Universal Robots PolyScope program: pick_place_robot_2.urp

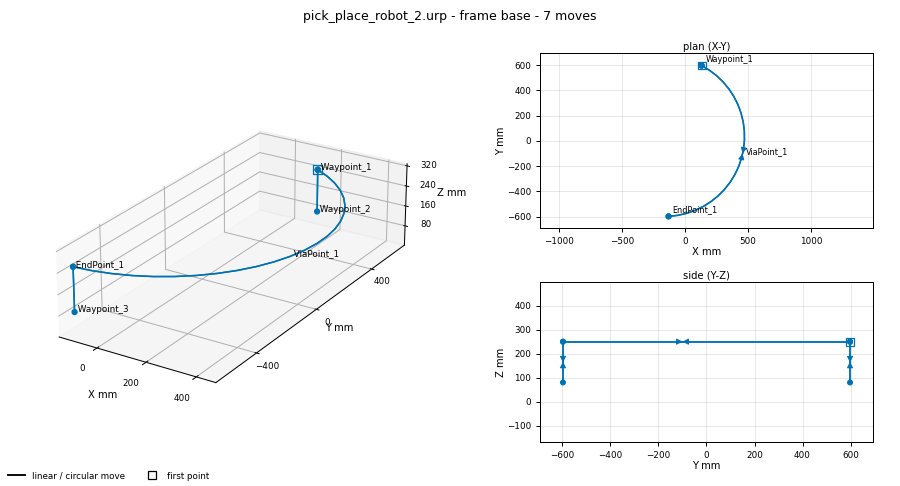
[picture p0: tool path of pick_place_robot_2.urp in frame base, 7 of 9 moves have a stored position in this frame; points joined in program order, loops and branches not executed]
Program pick_place_robot_2 (installation=default directory=/ursim/programs/new folder/new folder_1 createdIn=5.21.0 lastSavedIn=5.21.0 robotSerialNumber=20195599999)
Calibrated DH parameters: a=[0, -0.425, -0.3922, 0, 0, 0]; d=[0.1625, 0, 0, 0.1333, 0.0997, 0.0996]; alpha=[1.570796, 0, 0, 1.570796, -1.570796, 0]; deltaTheta=[0, 0, 0, 0, 0, 0]
InitVariablesNode
Robot Program (runOnlyOnce=false)
  MoveJ speed 60 deg/s, acceleration 80 deg/s^2 (useActiveTCP=true optimoveEnabled=false optiMoveSpeed=0.3 optiMoveAcceleration=0.09) feature=Base
    Waypoint Waypoint_1: TCP in base x=130.859 y=597.684 z=250 mm, rx=3.1159 ry=0.0355 rz=-0.0386 rad; joints [90, -112.778, -98.269, -60.415, 91.404, -1.323] deg; TCP offset x=0 y=0 z=0 mm, rx=0 ry=0 rz=0 rad
  Script: write_port_register(128,0)
  Script: write_port_register(160,0)
  Loop Forever
    Wait Sleep waitTime=0.5
    Script: write_port_register(128,1)
    Wait Condition expression=robot1set≟1
    Script: write_port_register(160,0)
    Script: write_port_register(128,0)
    Wait Condition expression=robot1ready≟1
    Script: write_port_register(160,1)
    MoveL speed 250 mm/s, acceleration 1200 mm/s^2 (useActiveTCP=true optimoveEnabled=false optiMoveSpeed=0.3 optiMoveAcceleration=0.09) feature=Base
      Waypoint Waypoint_2: TCP in base x=130.859 y=597.684 z=80 mm, rx=3.1159 ry=0.0355 rz=-0.0386 rad; joints [90, -128.474, -104.506, -38.481, 91.404, -1.323] deg; TCP offset x=0 y=0 z=0 mm, rx=0 ry=0 rz=0 rad
      Wait Sleep waitTime=1
      Waypoint Waypoint_1: TCP in base x=130.859 y=597.684 z=250 mm, rx=3.1159 ry=0.0355 rz=-0.0386 rad; joints [90, -112.778, -98.269, -60.415, 91.404, -1.323] deg; TCP offset x=0 y=0 z=0 mm, rx=0 ry=0 rz=0 rad
    Wait Sleep waitTime=0.5
    MoveP speed 250 mm/s, acceleration 1200 mm/s^2 (blendRadius=0.025 useActiveTCP=true optimoveEnabled=false optiMoveSpeed=0.3 optiMoveAcceleration=0.09) feature=Base
      CircleMove (OrientationMode=FIXED)
        Waypoint ViaPoint_1: TCP in base x=449.152 y=-130.859 z=250 mm, rx=2.246 ry=-2.1954 rz=-0.0556 rad; joints [0, -95.011, -121.58, -54.87, 91.404, -1.323] deg
        Waypoint EndPoint_1: TCP in base x=-130.859 y=-597.684 z=250 mm, rx=-0.0355 ry=3.1163 rz=0.0393 rad; joints [-90, -112.778, -98.269, -60.415, 91.404, -1.323] deg; TCP offset x=0 y=0 z=0 mm, rx=0 ry=0 rz=0 rad
    Wait Sleep waitTime=0.5
    MoveL speed 250 mm/s, acceleration 1200 mm/s^2 (useActiveTCP=true optimoveEnabled=false optiMoveSpeed=0.3 optiMoveAcceleration=0.09) feature=Base
      Waypoint Waypoint_3: TCP in base x=-130.859 y=-597.684 z=80 mm, rx=-0.0355 ry=3.1163 rz=0.0393 rad; joints [-90, -128.474, -104.506, -38.481, 91.404, -1.323] deg; TCP offset x=0 y=0 z=0 mm, rx=0 ry=0 rz=0 rad
      Wait Sleep waitTime=1
      Waypoint EndPoint_1: TCP in base x=-130.859 y=-597.684 z=250 mm, rx=-0.0355 ry=3.1163 rz=0.0393 rad; joints [-90, -112.778, -98.269, -60.415, 91.404, -1.323] deg; TCP offset x=0 y=0 z=0 mm, rx=0 ry=0 rz=0 rad
    Wait Sleep waitTime=0.5
    MoveP speed 250 mm/s, acceleration 1200 mm/s^2 (blendRadius=0.025 useActiveTCP=true optimoveEnabled=false optiMoveSpeed=0.3 optiMoveAcceleration=0.09) feature=Base
      CircleMove (OrientationMode=FIXED)
        Waypoint ViaPoint_1: TCP in base x=449.152 y=-130.859 z=250 mm, rx=2.246 ry=-2.1954 rz=-0.0556 rad; joints [0, -95.011, -121.58, -54.87, 91.404, -1.323] deg
        Waypoint Waypoint_1: TCP in base x=130.859 y=597.684 z=250 mm, rx=3.1159 ry=0.0355 rz=-0.0386 rad; joints [90, -112.778, -98.269, -60.415, 91.404, -1.323] deg; TCP offset x=0 y=0 z=0 mm, rx=0 ry=0 rz=0 rad
